// TIA Portal V19 export
TYPE "_EV_DataUDT"
   STRUCT
      "b" : Array[0..9] of Byte;
   END_STRUCT;
END_TYPE
